% RSLogix 500 project REV AND FOR_BAK006.RSS, saved by version 8.30.00.16 %
PROJECT "REV"    % processor: Bul.1763 MicroLogix 1100 Series B %

PROGRAM FILES
  LAD 2   3 rungs

DATA FILES
  O0 OUTPUT  4 elements
  I1 INPUT  6 elements
  S2 STATUS  66 elements
  B3 BINARY  1 elements
  T4 TIMER  1 elements
  C5 COUNTER  1 elements
  R6 CONTROL  1 elements
  N7 INTEGER  1 elements
  F8 FLOAT  1 elements

LADDER 2
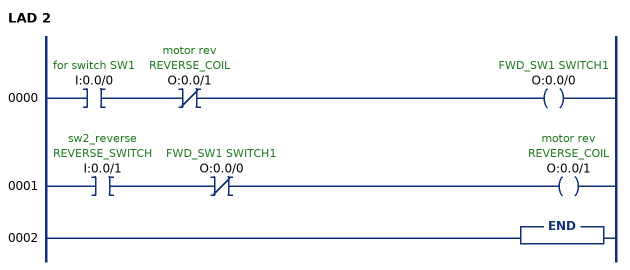
% Rung: 0 %
SOR XIC I:0.0/0 XIO O:0.0/1 OTE O:0.0/0 EOR
%   I:0.0/0  SW1  "for switch" %
%   O:0.0/1  REVERSE_COIL  "motor rev" %
%   O:0.0/0  SWITCH1  "FWD_SW1" %
% Rung: 1 %
SOR XIC I:0.0/1 XIO O:0.0/0 OTE O:0.0/1 EOR
%   I:0.0/1  REVERSE_SWITCH  "sw2_reverse" %
%   O:0.0/0  SWITCH1  "FWD_SW1" %
%   O:0.0/1  REVERSE_COIL  "motor rev" %
% Rung: 2 %
SOR END EOR
